(*
Limits the rate of change of the input signal.

The output tracks the input but cannot change faster than :attr:`RisingLimit`
units per second when increasing, or :attr:`FallingLimit` units per second when
decreasing. A limit of zero removes the restriction in that direction, allowing
the output to change freely.

Calling :meth:`Reset` snaps the output to the current input immediately.

.. note::
   The block is ``FINAL`` and must be instantiated, not extended.
   Use ``FB_init`` to set :attr:`fRisingLimit` and :attr:`fFallingLimit` at
   declaration time.
*)
{attribute 'enable_dynamic_creation'}
{attribute 'no_explicit_call' := 'direct call for this function block is not allowed'}
FUNCTION_BLOCK FINAL FB_RateLimiter EXTENDS FB_SisoComponent
IMPLEMENTS FsCommon.I_Runnable, I_Resettable
VAR
	_fRisingLimit  : LREAL; // Maximum rate of increase in units per second. Zero means no limit.
	_fFallingLimit : LREAL; // Maximum rate of decrease in units per second. Zero means no limit.
END_VAR

(*
Gets or sets the maximum rate of decrease in units per second.

The output will not fall faster than this value regardless of how quickly
the input changes. A value of zero removes the falling limit entirely.
Values below zero are clamped to zero.
*)
PROPERTY FallingLimit : LREAL
GET
FallingLimit := THIS^._fFallingLimit;
END_GET
SET
THIS^._fFallingLimit := MAX(0, FallingLimit);
END_SET
END_PROPERTY

METHOD FB_init : BOOL
VAR_INPUT
	bInitRetains   : BOOL; // if TRUE, the retain variables are initialized (warm start / cold start)
	bInCopyCode    : BOOL;  // if TRUE, the instance afterwards gets moved into the copy code (online change)
	fRisingLimit   : LREAL; // Maximum rate of increase in units per second. Zero means no limit.
	fFallingLimit  : LREAL; // Maximum rate of decrease in units per second. Zero means no limit.
END_VAR
THIS^.RisingLimit  := fRisingLimit;
THIS^.FallingLimit := fFallingLimit;
END_METHOD

(* Snaps the output to the current input, bypassing the rate limit. *)
METHOD Reset
VAR_INPUT
END_VAR
THIS^._fOutput := THIS^._fInput;
END_METHOD

(*
Gets or sets the maximum rate of increase in units per second.

The output will not rise faster than this value regardless of how quickly
the input changes. A value of zero removes the rising limit entirely.
Values below zero are clamped to zero.
*)
PROPERTY RisingLimit : LREAL
GET
RisingLimit := THIS^._fRisingLimit;
END_GET
SET
THIS^._fRisingLimit := MAX(0, RisingLimit);
END_SET
END_PROPERTY

(*
Advances the rate limiter by one time step.

.. note::
   Must be called once per cycle on a single PLC task. If the measured cycle
   time is zero the method returns early without updating the output.
*)
METHOD Run
VAR_INST
	{attribute 'hide'}
	bInit       : BOOL := TRUE;
	{attribute 'hide'}
	fT          : LREAL;
	{attribute 'hide'}
	fbTaskCycle : FsCommon.FB_PlcTaskCycleChangeDetector(0);
END_VAR
VAR
	fDelta    	: LREAL;
	fMaxDelta 	: LREAL;
END_VAR
IF bInit THEN
	fT := TO_LREAL(FsCommon.F_GetCurrentTaskCycleTime()) / TO_LREAL(LTIME#1S);
	RETURN(bInit := fT <= 0);
	fbTaskCycle.TaskIndex := FsCommon.F_GetCurrentTaskIndex();
	THIS^._fOutput := THIS^._fInput;
	RETURN;
END_IF

RETURN(NOT fbTaskCycle.HasChanged);

THIS^._fRisingLimit  := MAX(0, THIS^._fRisingLimit);
THIS^._fFallingLimit := MAX(0, THIS^._fFallingLimit);

fDelta := THIS^._fInput - THIS^._fOutput;

IF fDelta > 0 AND THIS^._fRisingLimit > 0 THEN
	fMaxDelta      := THIS^._fRisingLimit * fT;
	THIS^._fOutput := THIS^._fOutput + MIN(fDelta, fMaxDelta);
ELSIF fDelta < 0 AND THIS^._fFallingLimit > 0 THEN
	fMaxDelta      := THIS^._fFallingLimit * fT;
	THIS^._fOutput := THIS^._fOutput - MIN(ABS(fDelta), fMaxDelta);
ELSE
	THIS^._fOutput := THIS^._fInput;
END_IF
END_METHOD

END_FUNCTION_BLOCK

(* stored: Version 1.1.0.1, ProductVersion 3.1.4024.15
   POU FB_RateLimiter: Id {6b187191-fd48-454b-b40e-513b4b660686}, SpecialFunc None
   Property FallingLimit: Id {65e3de27-3938-4479-9570-005cce6e0121}
   Get Get: Id {fa7e4be6-7f73-49ec-a010-f1ee3115bbdb}
   Set Set: Id {d1288e13-41e6-41a7-ac19-85cac747afff}
   Method FB_init: Id {cfac3fab-8989-4336-9069-c763a2c4a875}
   Method Reset: Id {be89a069-a758-4c55-b388-a32be8a697ea}
   Property RisingLimit: Id {17ef19ac-68d3-46b2-8146-676ebe295d3b}
   Get Get: Id {7345b42a-9953-469f-b139-3cc0c80b3c47}
   Set Set: Id {d7f82d16-00d7-4613-9d2b-ae8e801207a9}
   Method Run: Id {ddc327d3-e350-442a-a454-06a785db0079} *)
